// TIA Portal V18 export
FUNCTION "Block_2" : Void   // FC1, LAD
{ S7_Optimized_Access := 'TRUE' }
VERSION : 0.1
// stored: AutoNumber true, IsIECCheckEnabled false, SetENOAutomatically false, UDAEnableTagReadback false
   VAR_INPUT
      w1 : Bool;
   END_VAR
   VAR_OUTPUT
      w2 : Bool;
   END_VAR
BEGIN

REGION Network 1
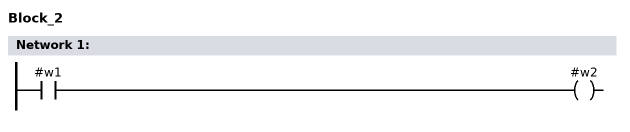
   RUNG wire#powerrail
      Contact( #w1 )
      Coil( #w2 )
   END_RUNG
   // the same network as SCL:
   #w2 := #w1;
END_REGION
END_FUNCTION
